    rq_wait_ft_sensor_steady(2000)
    zero_ftsensor()
    sleep(0.1)
    # end: URCap Program Node
    # begin: URCap Program Node
    #   Source: Robotiq_Copilot, 1.22.1.14215, Robotiq Inc.
    #   Type: Find Surface
    $ 164 "Find Surface"
    surface_found = rq_linear_search_urcap("Z+", 10.000, 0.005000, 0.100000, 1)
    storevar.setvariablepose("rq_findSurface_7514beb1-6ce4-4645-a4b6-934a629ef91f_exitPosition", get_actual_tcp_pose())
    $ 165 "'Add Stop conditions from the Find Surface node'" "noBreak"
    # 'Add Stop conditions from the Find Surface node'
    # end: URCap Program Node
    # begin: URCap Program Node
    #   Source: Robotiq_Copilot, 1.22.1.14215, Robotiq Inc.
    #   Type: Finishing Tool Control
    $ 166 "Start tool"
    set_standard_digital_out(0, True)
    # end: URCap Program Node
    $ 167 "Wait: 0.5"
    sleep(0.5)
    $ 168 "MoveL"
    $ 169 "Force"
    sleep(0.02)
    zero_ftsensor()
    force_mode(tool_pose(), [0, 0, 1, 0, 0, 0], [0.0, 0.0, 5.0, 0.0, 0.0, 0.0], 2, [0.1, 0.1, 0.15, 0.3490658503988659, 0.3490658503988659, 0.3490658503988659])
    $ 170 "Direction: CubeFront Y+" "noBreak"
    global move_thread_flag_170=0
    thread move_thread_170():
      enter_critical
      move_thread_flag_170 = 1
      local towardsPos=calculate_point_to_move_towards(p[0.009684890691344802,0.6183777132013698,0.176868741957311,1.5686992879971895,-0.013964727372415317,-0.007428573495752937], [0.0,1.0,0.0], 0.355)
      movel(towardsPos, a=1.2, v=0.06)
      move_thread_flag_170 = 2
      exit_critical
    end
    move_thread_flag_170 = 0
    move_thread_han_170 = run move_thread_170()
    while (True):
      sleep(1.0E-10)
      if (move_thread_flag_170 > 1):
        join move_thread_han_170
        $ 171 "Until (distance)" "noBreak"
        break
      end
      sync()
    end
    $ 172 "Direction: CubeFront X+" "noBreak"
    global move_thread_flag_172=0
    thread move_thread_172():
      enter_critical
      move_thread_flag_172 = 1
      local towardsPos=calculate_point_to_move_towards(p[0.009684890691344802,0.6183777132013698,0.176868741957311,1.5686992879971895,-0.013964727372415317,-0.007428573495752937], [1.0,0.0,0.0], 0.355)
      movel(towardsPos, a=1.2, v=0.06)
      move_thread_flag_172 = 2
      exit_critical
    end
    move_thread_flag_172 = 0
    move_thread_han_172 = run move_thread_172()
    while (True):
      sleep(1.0E-10)
      if (move_thread_flag_172 > 1):
        join move_thread_han_172
        $ 173 "Until (distance)" "noBreak"
        break
      end
      sync()
    end
    $ 174 "Direction: CubeFront Y-" "noBreak"
    global move_thread_flag_174=0
    thread move_thread_174():
      enter_critical
      move_thread_flag_174 = 1
      local towardsPos=calculate_point_to_move_towards(p[0.009684890691344802,0.6183777132013698,0.176868741957311,1.5686992879971895,-0.013964727372415317,-0.007428573495752937], [0.0,-1.0,0.0], 0.355)
      movel(towardsPos, a=1.2, v=0.06)
      move_thread_flag_174 = 2
      exit_critical
    end
    move_thread_flag_174 = 0
    move_thread_han_174 = run move_thread_174()
    while (True):
      sleep(1.0E-10)
      if (move_thread_flag_174 > 1):
        join move_thread_han_174
        $ 175 "Until (distance)" "noBreak"
        break
      end
      sync()
    end
    $ 176 "Direction: CubeFront X-" "noBreak"
    global move_thread_flag_176=0
    thread move_thread_176():
      enter_critical
      move_thread_flag_176 = 1
      local towardsPos=calculate_point_to_move_towards(p[0.009684890691344802,0.6183777132013698,0.176868741957311,1.5686992879971895,-0.013964727372415317,-0.007428573495752937], [-1.0,0.0,0.0], 0.355)
      movel(towardsPos, a=1.2, v=0.06)
      move_thread_flag_176 = 2
      exit_critical
    end
    move_thread_flag_176 = 0
    move_thread_han_176 = run move_thread_176()
    while (True):
      sleep(1.0E-10)
      if (move_thread_flag_176 > 1):
        join move_thread_han_176
        $ 177 "Until (distance)" "noBreak"
        break
      end
      sync()
    end
    # begin: URCap Program Node
    #   Source: Robotiq_Copilot, 1.22.1.14215, Robotiq Inc.
    #   Type: Finishing Tool Control
    $ 178 "Stop tool" "noBreak"
    set_standard_digital_out(0, False)
    # end: URCap Program Node
    end_force_mode()
    stopl(5.0)
    $ 179 "Direction: Tool Z-"
    global move_thread_flag_179=0
    thread move_thread_179():
      enter_critical
      move_thread_flag_179 = 1
      local towardsPos=calculate_point_to_move_towards(get_forward_kin(), [0.0,0.0,-1.0], 0.025)
      movel(towardsPos, a=1.2, v=0.06)
      move_thread_flag_179 = 2
      exit_critical
    end
    move_thread_flag_179 = 0
    move_thread_han_179 = run move_thread_179()
    while (True):
      sleep(1.0E-10)
      if (move_thread_flag_179 > 1):
        join move_thread_han_179
        $ 180 "Until (distance)"
        break
      end
      sync()
    end
    $ 181 "MoveJ"
    $ 182 "clear" "breakAfter"
    movej(clear_q, a=1.3962634015954636, v=1.0471975511965976)
  end
  def StartSpray():
    $ 183 "StartSpray" "noBreak"
    $ 184 "Set DO[1]=On"
    set_standard_digital_out(1, True)
    $ 185 "Wait: 0.3"
    sleep(0.3)
  end
  def stopSpray():
    $ 186 "stopSpray" "noBreak"
    $ 187 "Set DO[1]=Off"
    set_standard_digital_out(1, False)
    $ 188 "Wait: 0.3"
    sleep(0.3)
  end
  thread EventThread():
    while (True):
      if (get_standard_digital_in(1) !=   True  ):
        $ 54 "Set DO[0]=Off"
        set_standard_digital_out(0, False)
        $ 55 "Set DO[1]=Off"
        set_standard_digital_out(1, False)
        $ 56 "Halt"
        halt
      end
      sync()
    end
  end
  eventThread = run EventThread()
  while (True):
    $ 1 "Robot Program"
    $ 2 "Main"
    $ 3 "MoveJ"
    $ 4 "clear" "breakAfter"
    movej(clear_q, a=1.3962634015954636, v=1.0471975511965976)
    # begin: URCap Program Node
    #   Source: Robotiq_Copilot, 1.22.1.14215, Robotiq Inc.
    #   Type: Zero FT Sensor
    $ 5 "Zero FT Sensor"

    rq_wait_ft_sensor_steady(2000)
    zero_ftsensor()
    sleep(0.1)
    # end: URCap Program Node
    $ 6 "Wait DI[0]=HI"
    while (get_standard_digital_in(0) == False):
      sync()
    end
    $ 7 "Call SandFront"
    SandFront()
    $ 8 "Call SandFront"
    SandFront()
    $ 9 "Call SandRebate"
    SandRebate()
    $ 10 "Call SandRebate"
    SandRebate()
    $ 11 "Wait DI[0]=HI"
    while (get_standard_digital_in(0) == False):
      sync()
    end
    $ 12 "Call SprayFront"
    SprayFront()
    $ 13 "Call SprayFront"
    SprayFront()
    $ 14 "Call SprayRebate"
    SprayRebate()
    $ 15 "Call SprayRebate"
    SprayRebate()
    $ 16 "Wait DI[0]=HI"
    while (get_standard_digital_in(0) == False):
      sync()
    end
    $ 17 "Call SandFront"
    SandFront()
    $ 18 "Call SandFront"
    SandFront()
  end
end
